FUNCTION_BLOCK OF_E_RTimeOut (* Simple implementation of the timeout services *)
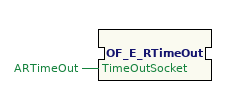
  SOCKETS
    TimeOutSocket : iec61499::events::ARTimeOut;
  END_SOCKETS
END_FUNCTION_BLOCK
